# EPICS substitutions: ATTOCUBE/ATTOCUBE-IOC-01App/Db/common.substitutions
file $(ATTOCUBE)/db/ancController.template {
pattern
{P,   PORT}
{\$(P), \$(PORT)}
}
